// TIA Portal V20 export
// export: Created 2025-12-01T14:57:21.2984252Z, ExportSetting None, DisplayName Totally Integrated Automation Portal, DisplayVersion V20 Update 3, DisplayName TIA Portal Openness, DisplayVersion V20 Update 3, DisplayName TIA Portal Version Control Interface, DisplayVersion V20 Update 3, DisplayName STEP 7 Professional, DisplayVersion V20 Update 3, DisplayName STEP 7 Safety, DisplayVersion V20 Update 2, DisplayName WinCC Basic/Comfort/Advanced, DisplayVersion V20 Update 3, DisplayName WinCC Professional, DisplayVersion V20 Update 3, DisplayName WinCC Unified, DisplayVersion V20 Update 3
FUNCTION "FC2002_SeguridadesAuxiliares" : Void   // FC2002, LAD
TITLE = Seguridades Auxiliares
{ S7_Optimized_Access := 'FALSE' }
// poner cada señal de sinoptico puesta en el FC2001 a que armario de potencia y 
// linea pertenece
// stored: AutoNumber false, SetENOAutomatically false
   VAR_TEMP
      basura : Int;
      TEMPWORD : Word;
      ESTRUCTURA AT TEMPWORD : Array[0..15] of Bool;
   END_VAR
BEGIN

REGION Network 1: Sinoptico Setas de Emergencia
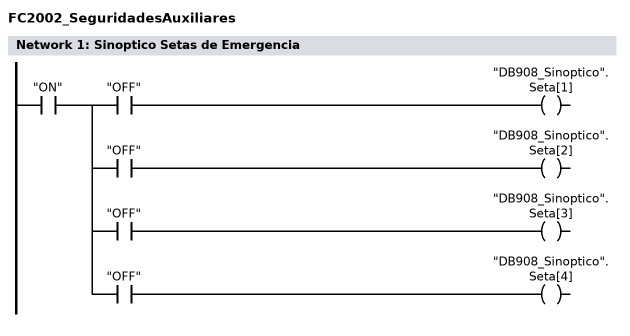
   RUNG wire#powerrail
      Contact( "ON" )
      wire#w1
      Contact( "OFF" )
      Coil( "DB908_Sinoptico".Seta[1] )
   END_RUNG
   RUNG wire#w1
      Contact( "OFF" )
      Coil( "DB908_Sinoptico".Seta[2] )
   END_RUNG
   RUNG wire#w1
      Contact( "OFF" )
      Coil( "DB908_Sinoptico".Seta[3] )
   END_RUNG
   RUNG wire#w1
      Contact( "OFF" )
      Coil( "DB908_Sinoptico".Seta[4] )
   END_RUNG
   // the same network as SCL:
   "DB908_Sinoptico".Seta[1] := "ON" AND "OFF";
   "DB908_Sinoptico".Seta[2] := "ON" AND "OFF";
   "DB908_Sinoptico".Seta[3] := "ON" AND "OFF";
   "DB908_Sinoptico".Seta[4] := "ON" AND "OFF";
END_REGION
END_FUNCTION
